// TIA Portal V18 export
VAR_GLOBAL   // PLC tag table "Cabinet_8"
   Sz8_Button_LED_ST06_ST07 AT %Q1800.0 : Bool;
   Sz8_Button_LED_ST07_ST08 AT %Q1800.1 : Bool;
   Sz8_Button_LED_ST08_ST09 AT %Q1800.2 : Bool;
   Sz8_Button_LED_Centering_ST08 AT %Q1800.3 : Bool;
   "Reserved(108)" AT %Q1800.4 : Bool;
   "Reserved(109)" AT %Q1800.5 : Bool;
   "Reserved(110)" AT %Q1800.6 : Bool;
   "Reserved(111)" AT %Q1800.7 : Bool;
   Sz8_ST06_SenA AT %I1800.0 : Bool;
   Sz8_ST06_SenB AT %I1800.1 : Bool;
   Sz8_ST06_SenC AT %I1800.2 : Bool;
   Sz8_ST06_SenD AT %I1800.3 : Bool;
   Sz8_ST07_SenA AT %I1800.4 : Bool;
   Sz8_ST07_SenB AT %I1800.5 : Bool;
   Sz8_ST07_SenC AT %I1800.6 : Bool;
   Sz8_ST07_SenD AT %I1800.7 : Bool;
   Sz8_ST08_SenA AT %I1801.0 : Bool;
   Sz8_ST08_SenB AT %I1801.1 : Bool;
   Sz8_ST08_SenC AT %I1801.2 : Bool;
   Sz8_ST08_SenD AT %I1801.3 : Bool;
   Sz8_Button_ST06_ST07 AT %I1801.4 : Bool;
   Sz8_Button_ST07_ST08 AT %I1801.5 : Bool;
   Sz8_Button_ST08_ST09 AT %I1801.6 : Bool;
   Sz8_Button_Centering_ST08 AT %I1801.7 : Bool;
   Sz8_Safety1_1 AT %I1850.0 : Bool;
   "Reserved(112)" AT %I1850.1 : Bool;
   "Reserved(113)" AT %I1850.2 : Bool;
   "Reserved(114)" AT %I1850.3 : Bool;
   Sz8_Safety1_2 AT %I1850.4 : Bool;
   "Reserved(115)" AT %I1850.5 : Bool;
   "Reserved(116)" AT %I1850.6 : Bool;
   "Reserved(117)" AT %I1850.7 : Bool;
   "Reserved(118)" AT %I1851.0 : Bool;
   "Reserved(119)" AT %I1851.1 : Bool;
   "Reserved(120)" AT %I1851.2 : Bool;
   "Reserved(121)" AT %I1851.3 : Bool;
   "Reserved(122)" AT %I1851.4 : Bool;
   "Reserved(123)" AT %I1851.5 : Bool;
   "Reserved(124)" AT %I1851.6 : Bool;
   "Reserved(125)" AT %I1851.7 : Bool;
END_VAR
